# EPICS autosave request: autosave/galil_digital_out_bit.req
$(P)$(R)_CMD
